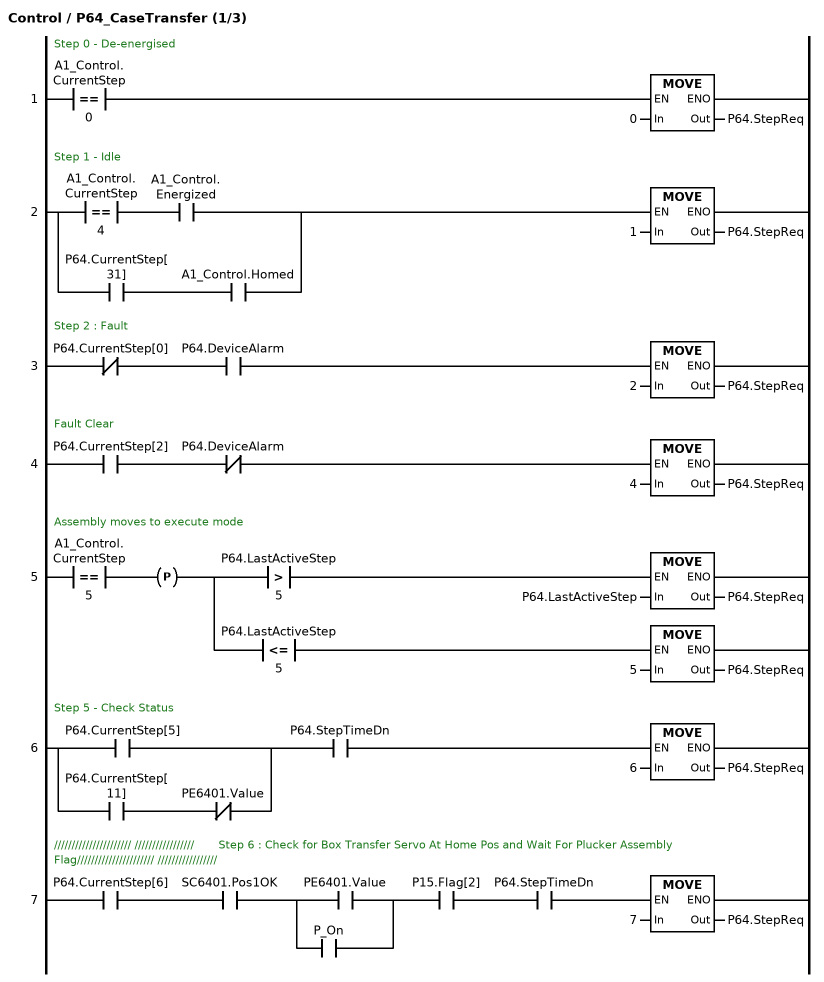
(* [picture p24: Control / P64_CaseTransfer, rungs 1-7] *)
(* Rung 1: Step 0 - De-energised *)
IF A1_Control.CurrentStep = 0 THEN P64.StepReq := 0; END_IF;
(* Rung 2: Step 1 - Idle *)
IF ((A1_Control.CurrentStep = 4) AND A1_Control.Energized) OR (P64.CurrentStep[31] AND A1_Control.Homed) THEN
    P64.StepReq := 1;
END_IF;
(* Rung 3: Step 2 : Fault *)
IF NOT P64.CurrentStep[0] AND P64.DeviceAlarm THEN P64.StepReq := 2; END_IF;
(* Rung 4: Fault Clear *)
IF P64.CurrentStep[2] AND NOT P64.DeviceAlarm THEN P64.StepReq := 4; END_IF;
(* Rung 5: Assembly moves to execute mode *)
_e10(CLK := A1_Control.CurrentStep = 5);
IF _e10.Q AND (P64.LastActiveStep > 5) THEN P64.StepReq := P64.LastActiveStep; END_IF;
IF _e10.Q AND (P64.LastActiveStep <= 5) THEN P64.StepReq := 5; END_IF;
(* Rung 6: Step 5 - Check Status *)
IF (P64.CurrentStep[5] OR (P64.CurrentStep[11] AND NOT PE6401.Value)) AND P64.StepTimeDn THEN
    P64.StepReq := 6;
END_IF;
(* Rung 7: ////////////////////// /////////////////       Step 6 : Check for Box Transfer Servo At Home Pos and Wait For Plucker Assembly Flag////////////////////// ///////////////// *)
IF P64.CurrentStep[6] AND SC6401.Pos1OK AND (PE6401.Value OR P_On) AND P15.Flag[2] AND P64.StepTimeDn THEN
    P64.StepReq := 7;
END_IF;

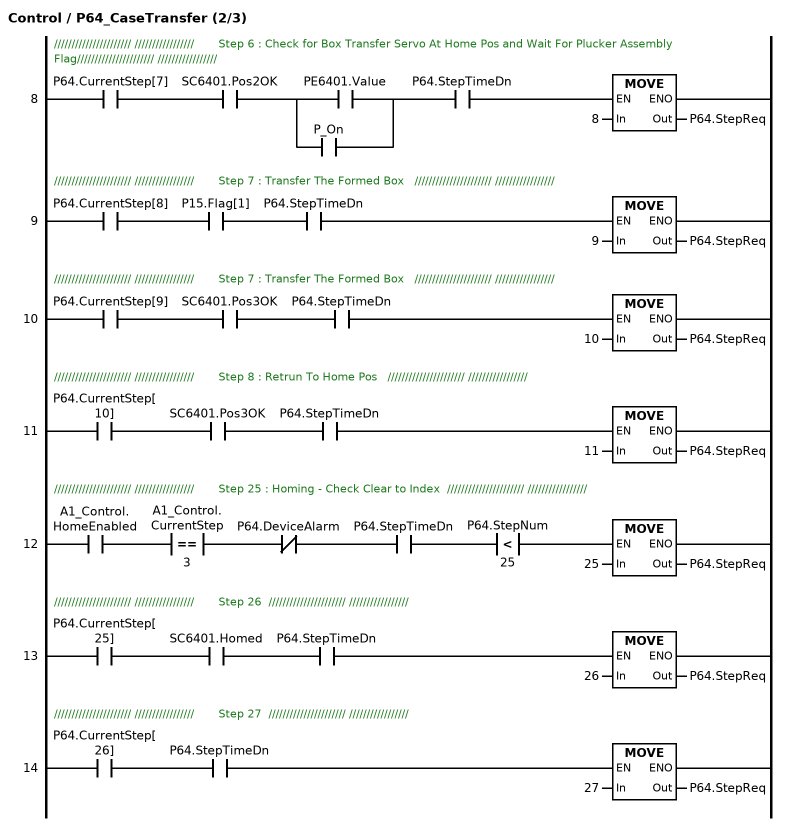
(* Rung 8: ////////////////////// /////////////////       Step 6 : Check for Box Transfer Servo At Home Pos and Wait For Plucker Assembly Flag////////////////////// ///////////////// *)
IF P64.CurrentStep[7] AND SC6401.Pos2OK AND (PE6401.Value OR P_On) AND P64.StepTimeDn THEN
    P64.StepReq := 8;
END_IF;
(* Rung 9: ////////////////////// /////////////////       Step 7 : Transfer The Formed Box   ////////////////////// ///////////////// *)
IF P64.CurrentStep[8] AND P15.Flag[1] AND P64.StepTimeDn THEN P64.StepReq := 9; END_IF;
(* Rung 10: ////////////////////// /////////////////       Step 7 : Transfer The Formed Box   ////////////////////// ///////////////// *)
IF P64.CurrentStep[9] AND SC6401.Pos3OK AND P64.StepTimeDn THEN P64.StepReq := 10; END_IF;
(* Rung 11: ////////////////////// /////////////////       Step 8 : Retrun To Home Pos   ////////////////////// ///////////////// *)
IF P64.CurrentStep[10] AND SC6401.Pos3OK AND P64.StepTimeDn THEN P64.StepReq := 11; END_IF;
(* Rung 12: ////////////////////// /////////////////       Step 25 : Homing - Check Clear to Index  ////////////////////// ///////////////// *)
IF A1_Control.HomeEnabled AND (A1_Control.CurrentStep = 3) AND NOT P64.DeviceAlarm AND P64.StepTimeDn AND (P64.StepNum < 25) THEN
    P64.StepReq := 25;
END_IF;
(* Rung 13: ////////////////////// /////////////////       Step 26  ////////////////////// ///////////////// *)
IF P64.CurrentStep[25] AND SC6401.Homed AND P64.StepTimeDn THEN P64.StepReq := 26; END_IF;
(* Rung 14: ////////////////////// /////////////////       Step 27  ////////////////////// ///////////////// *)
IF P64.CurrentStep[26] AND P64.StepTimeDn THEN P64.StepReq := 27; END_IF;

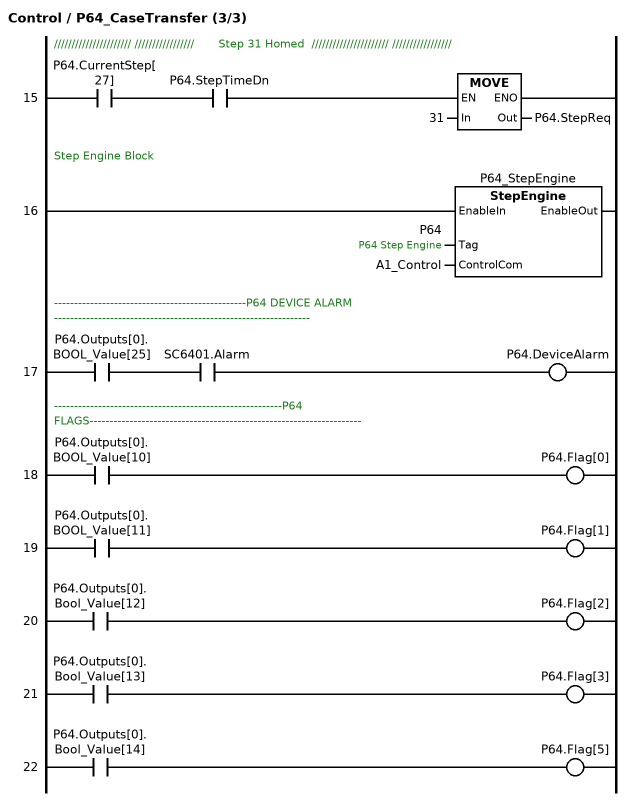
(* Rung 15: ////////////////////// /////////////////       Step 31 Homed  ////////////////////// ///////////////// *)
IF P64.CurrentStep[27] AND P64.StepTimeDn THEN P64.StepReq := 31; END_IF;
(* Rung 16: Step Engine Block *)
P64_StepEngine(EnableIn := TRUE, Tag := P64, ControlCom := A1_Control);
(* Rung 17: ------------------------------------------------P64 DEVICE ALARM ---------------------------------------------------------------- *)
P64.DeviceAlarm := P64.Outputs[0].BOOL_Value[25] AND SC6401.Alarm;
(* Rung 18: ---------------------------------------------------------P64 FLAGS-------------------------------------------------------------------- *)
P64.Flag[0] := P64.Outputs[0].BOOL_Value[10];
(* Rung 19 *)
P64.Flag[1] := P64.Outputs[0].BOOL_Value[11];
(* Rung 20 *)
P64.Flag[2] := P64.Outputs[0].Bool_Value[12];
(* Rung 21 *)
P64.Flag[3] := P64.Outputs[0].Bool_Value[13];
(* Rung 22 *)
P64.Flag[5] := P64.Outputs[0].Bool_Value[14];

(* Section P22_BottomTaping: ladder, written here as Structured Text *)

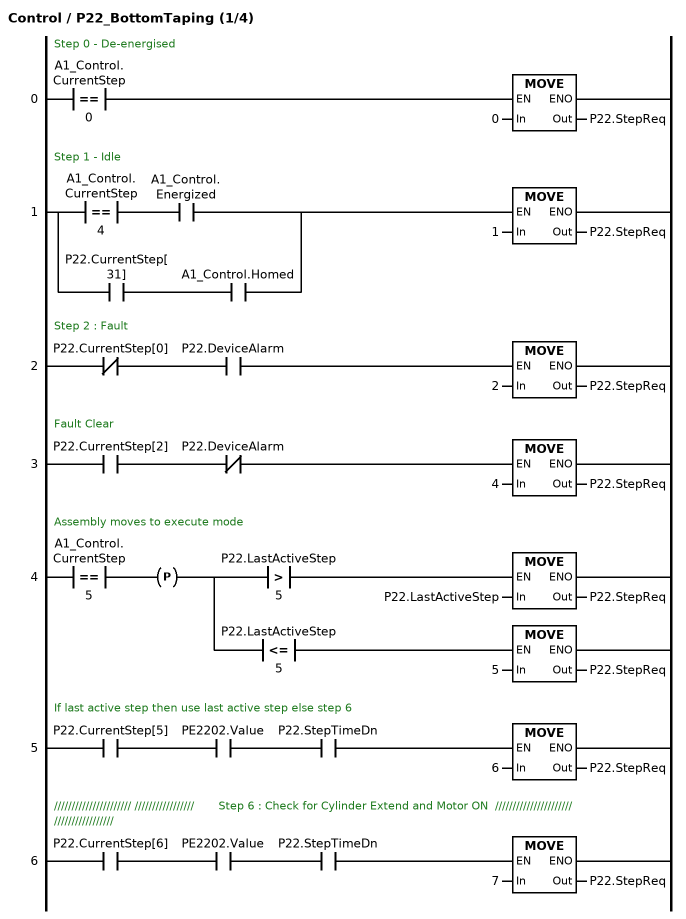
(* Rung 0: Step 0 - De-energised *)
IF A1_Control.CurrentStep = 0 THEN P22.StepReq := 0; END_IF;
(* Rung 1: Step 1 - Idle *)
IF ((A1_Control.CurrentStep = 4) AND A1_Control.Energized) OR (P22.CurrentStep[31] AND A1_Control.Homed) THEN
    P22.StepReq := 1;
END_IF;
(* Rung 2: Step 2 : Fault *)
IF NOT P22.CurrentStep[0] AND P22.DeviceAlarm THEN P22.StepReq := 2; END_IF;
(* Rung 3: Fault Clear *)
IF P22.CurrentStep[2] AND NOT P22.DeviceAlarm THEN P22.StepReq := 4; END_IF;
(* Rung 4: Assembly moves to execute mode *)
_e11(CLK := A1_Control.CurrentStep = 5);
IF _e11.Q AND (P22.LastActiveStep > 5) THEN P22.StepReq := P22.LastActiveStep; END_IF;
IF _e11.Q AND (P22.LastActiveStep <= 5) THEN P22.StepReq := 5; END_IF;
(* Rung 5: If last active step then use last active step else step 6 *)
IF P22.CurrentStep[5] AND PE2202.Value AND P22.StepTimeDn THEN P22.StepReq := 6; END_IF;
(* Rung 6: ////////////////////// /////////////////       Step 6 : Check for Cylinder Extend and Motor ON  ////////////////////// ///////////////// *)
IF P22.CurrentStep[6] AND PE2202.Value AND P22.StepTimeDn THEN P22.StepReq := 7; END_IF;

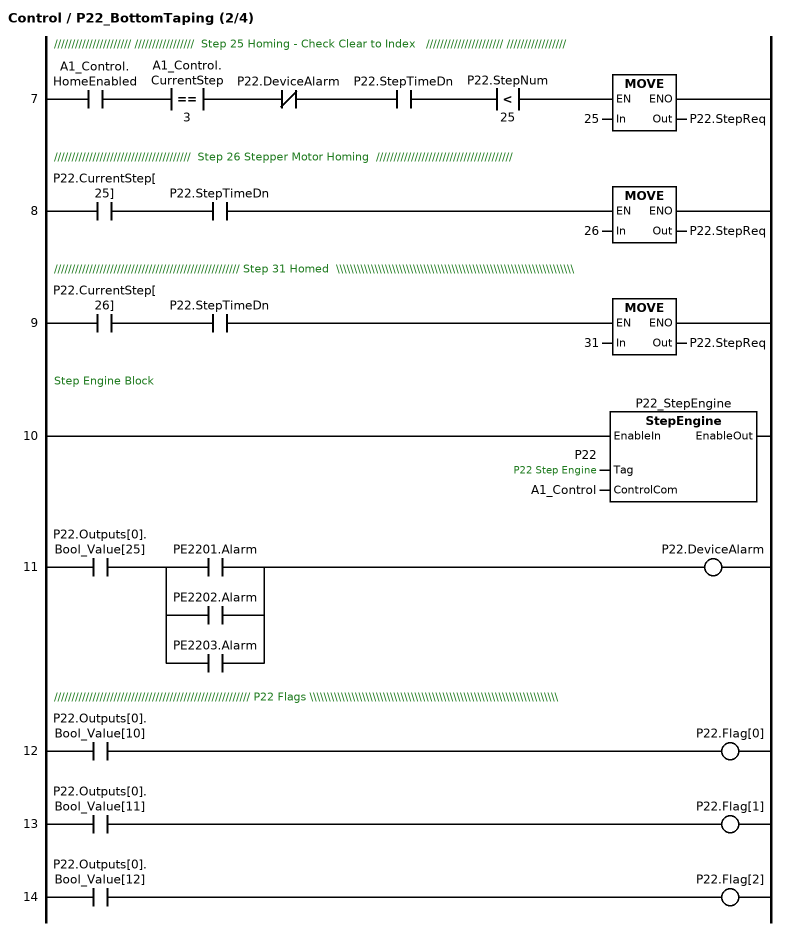
(* Rung 7: ////////////////////// /////////////////  Step 25 Homing - Check Clear to Index   ////////////////////// ///////////////// *)
IF A1_Control.HomeEnabled AND (A1_Control.CurrentStep = 3) AND NOT P22.DeviceAlarm AND P22.StepTimeDn AND (P22.StepNum < 25) THEN
    P22.StepReq := 25;
END_IF;
(* Rung 8: ///////////////////////////////////////  Step 26 Stepper Motor Homing  /////////////////////////////////////// *)
IF P22.CurrentStep[25] AND P22.StepTimeDn THEN P22.StepReq := 26; END_IF;
(* Rung 9: ///////////////////////////////////////////////////// Step 31 Homed  \\\\\\\\\\\\\\\\\\\\\\\\\\\\\\\\\\\\\\\\\\\\\\\\\\\\\\\\\\\\\\\\\\\\ *)
IF P22.CurrentStep[26] AND P22.StepTimeDn THEN P22.StepReq := 31; END_IF;
(* Rung 10: Step Engine Block *)
P22_StepEngine(EnableIn := TRUE, Tag := P22, ControlCom := A1_Control);
(* Rung 11 *)
P22.DeviceAlarm := P22.Outputs[0].Bool_Value[25] AND (PE2201.Alarm OR PE2202.Alarm OR PE2203.Alarm);
(* Rung 12: //////////////////////////////////////////////////////// P22 Flags \\\\\\\\\\\\\\\\\\\\\\\\\\\\\\\\\\\\\\\\\\\\\\\\\\\\\\\\\\\\\\\\\\\\\\\ *)
P22.Flag[0] := P22.Outputs[0].Bool_Value[10];
(* Rung 13 *)
P22.Flag[1] := P22.Outputs[0].Bool_Value[11];
(* Rung 14 *)
P22.Flag[2] := P22.Outputs[0].Bool_Value[12];

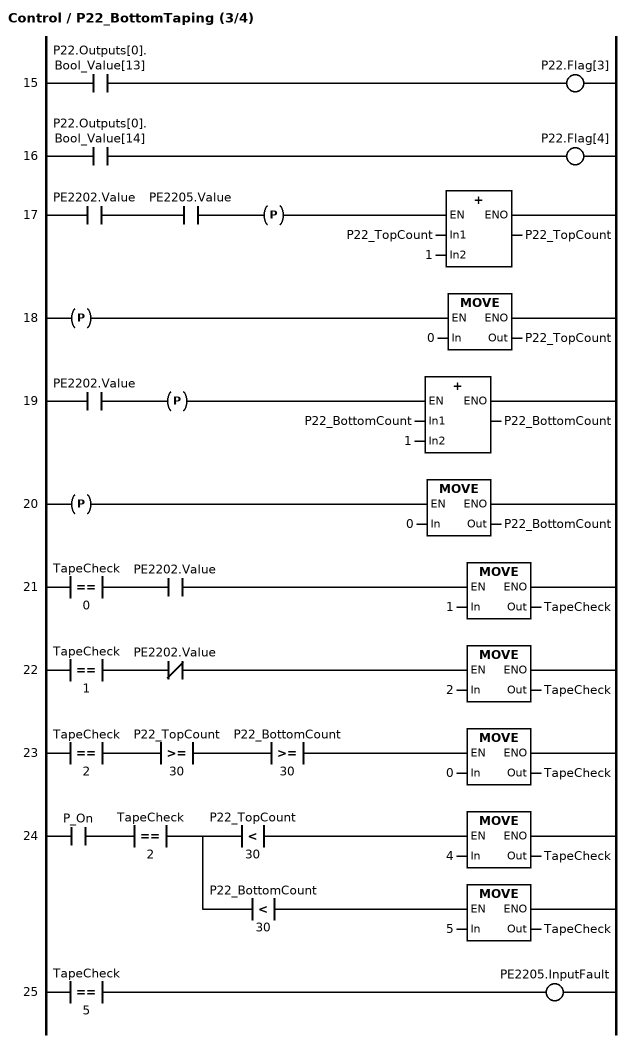
(* Rung 15 *)
P22.Flag[3] := P22.Outputs[0].Bool_Value[13];
(* Rung 16 *)
P22.Flag[4] := P22.Outputs[0].Bool_Value[14];
(* Rung 17 *)
_e12(CLK := PE2202.Value AND PE2205.Value);
IF _e12.Q THEN P22_TopCount := P22_TopCount + 1; END_IF;
(* Rung 18 *)
_e13(CLK := TRUE);
IF _e13.Q THEN P22_TopCount := 0; END_IF;
(* Rung 19 *)
_e14(CLK := PE2202.Value);
IF _e14.Q THEN P22_BottomCount := P22_BottomCount + 1; END_IF;
(* Rung 20 *)
_e15(CLK := TRUE);
IF _e15.Q THEN P22_BottomCount := 0; END_IF;
(* Rung 21 *)
IF (TapeCheck = 0) AND PE2202.Value THEN TapeCheck := 1; END_IF;
(* Rung 22 *)
IF (TapeCheck = 1) AND NOT PE2202.Value THEN TapeCheck := 2; END_IF;
(* Rung 23 *)
IF (TapeCheck = 2) AND (P22_TopCount >= 30) AND (P22_BottomCount >= 30) THEN TapeCheck := 0; END_IF;
(* Rung 24 *)
_p16 := P_On AND (TapeCheck = 2);
IF P_On AND (TapeCheck = 2) AND (P22_TopCount < 30) THEN TapeCheck := 4; END_IF;
IF _p16 AND (P22_BottomCount < 30) THEN TapeCheck := 5; END_IF;
(* Rung 25 *)
PE2205.InputFault := TapeCheck = 5;

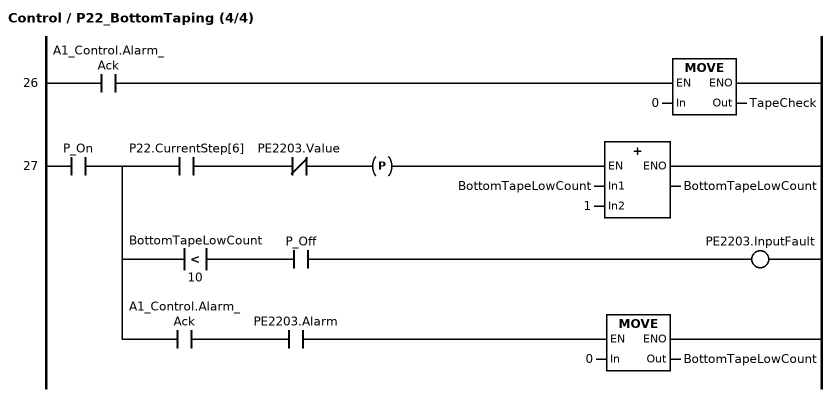
(* Rung 26 *)
IF A1_Control.Alarm_Ack THEN TapeCheck := 0; END_IF;
(* Rung 27 *)
_e17(CLK := P_On AND P22.CurrentStep[6] AND NOT PE2203.Value);
IF _e17.Q THEN BottomTapeLowCount := BottomTapeLowCount + 1; END_IF;
PE2203.InputFault := P_On AND (BottomTapeLowCount < 10) AND P_Off;
IF P_On AND A1_Control.Alarm_Ack AND PE2203.Alarm THEN BottomTapeLowCount := 0; END_IF;

(* Section P18_InfeedConveyor_1: ladder, written here as Structured Text *)

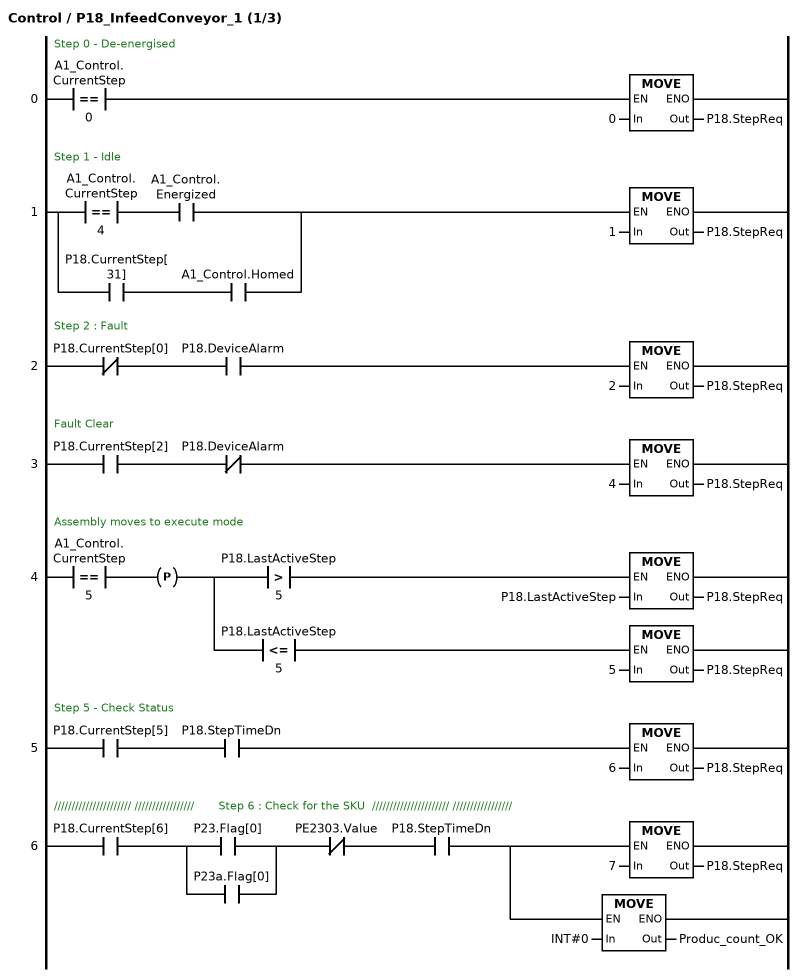
(* Rung 0: Step 0 - De-energised *)
IF A1_Control.CurrentStep = 0 THEN P18.StepReq := 0; END_IF;
(* Rung 1: Step 1 - Idle *)
IF ((A1_Control.CurrentStep = 4) AND A1_Control.Energized) OR (P18.CurrentStep[31] AND A1_Control.Homed) THEN
    P18.StepReq := 1;
END_IF;
(* Rung 2: Step 2 : Fault *)
IF NOT P18.CurrentStep[0] AND P18.DeviceAlarm THEN P18.StepReq := 2; END_IF;
(* Rung 3: Fault Clear *)
IF P18.CurrentStep[2] AND NOT P18.DeviceAlarm THEN P18.StepReq := 4; END_IF;
(* Rung 4: Assembly moves to execute mode *)
_e18(CLK := A1_Control.CurrentStep = 5);
IF _e18.Q AND (P18.LastActiveStep > 5) THEN P18.StepReq := P18.LastActiveStep; END_IF;
IF _e18.Q AND (P18.LastActiveStep <= 5) THEN P18.StepReq := 5; END_IF;
(* Rung 5: Step 5 - Check Status *)
IF P18.CurrentStep[5] AND P18.StepTimeDn THEN P18.StepReq := 6; END_IF;
(* Rung 6: ////////////////////// /////////////////       Step 6 : Check for the SKU  ////////////////////// ///////////////// *)
_p19 := P18.CurrentStep[6] AND (P23.Flag[0] OR P23a.Flag[0]) AND NOT PE2303.Value AND P18.StepTimeDn;
IF _p19 THEN
    P18.StepReq := 7;
    Produc_count_OK := INT#0;
END_IF;

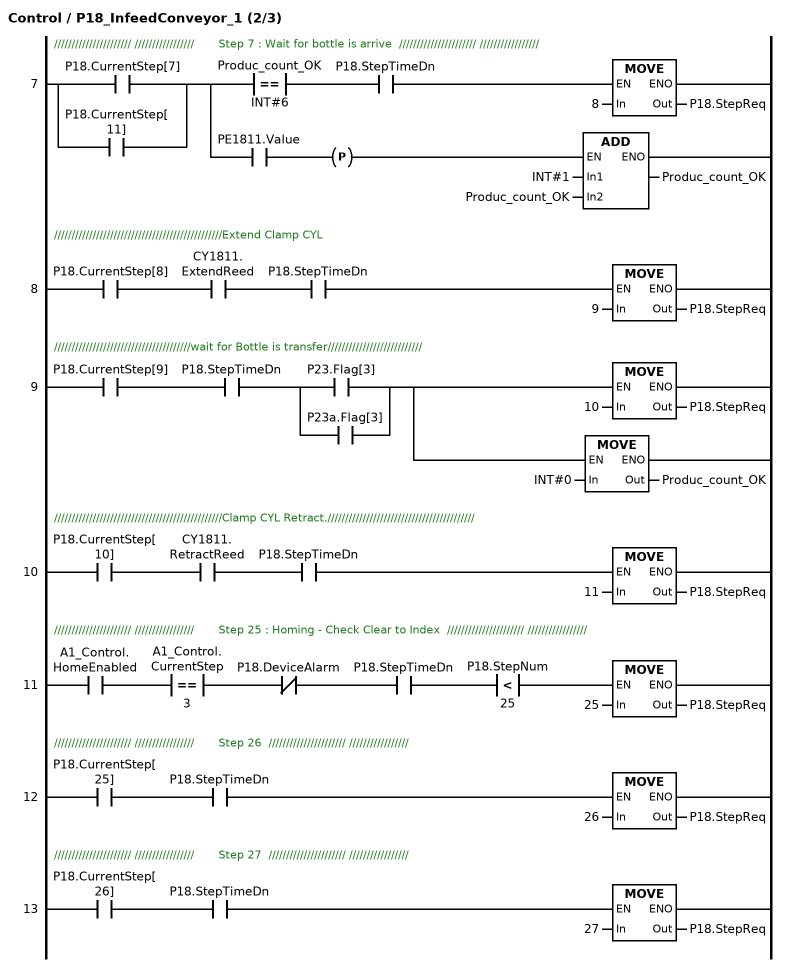
(* Rung 7: ////////////////////// /////////////////       Step 7 : Wait for bottle is arrive  ////////////////////// ///////////////// *)
_p20 := P18.CurrentStep[7] OR P18.CurrentStep[11];
IF (P18.CurrentStep[7] OR P18.CurrentStep[11]) AND (Produc_count_OK = INT#6) AND P18.StepTimeDn THEN
    P18.StepReq := 8;
END_IF;
_e21(CLK := _p20 AND PE1811.Value);
IF _e21.Q THEN Produc_count_OK := INT#1 + Produc_count_OK; END_IF;
(* Rung 8: ////////////////////////////////////////////////Extend Clamp CYL *)
IF P18.CurrentStep[8] AND CY1811.ExtendReed AND P18.StepTimeDn THEN P18.StepReq := 9; END_IF;
(* Rung 9: ///////////////////////////////////////wait for Bottle is transfer/////////////////////////// *)
_p22 := P18.CurrentStep[9] AND P18.StepTimeDn AND (P23.Flag[3] OR P23a.Flag[3]);
IF _p22 THEN
    P18.StepReq := 10;
    Produc_count_OK := INT#0;
END_IF;
(* Rung 10: ////////////////////////////////////////////////Clamp CYL Retract.////////////////////////////////////////// *)
IF P18.CurrentStep[10] AND CY1811.RetractReed AND P18.StepTimeDn THEN P18.StepReq := 11; END_IF;
(* Rung 11: ////////////////////// /////////////////       Step 25 : Homing - Check Clear to Index  ////////////////////// ///////////////// *)
IF A1_Control.HomeEnabled AND (A1_Control.CurrentStep = 3) AND NOT P18.DeviceAlarm AND P18.StepTimeDn AND (P18.StepNum < 25) THEN
    P18.StepReq := 25;
END_IF;
(* Rung 12: ////////////////////// /////////////////       Step 26  ////////////////////// ///////////////// *)
IF P18.CurrentStep[25] AND P18.StepTimeDn THEN P18.StepReq := 26; END_IF;
(* Rung 13: ////////////////////// /////////////////       Step 27  ////////////////////// ///////////////// *)
IF P18.CurrentStep[26] AND P18.StepTimeDn THEN P18.StepReq := 27; END_IF;

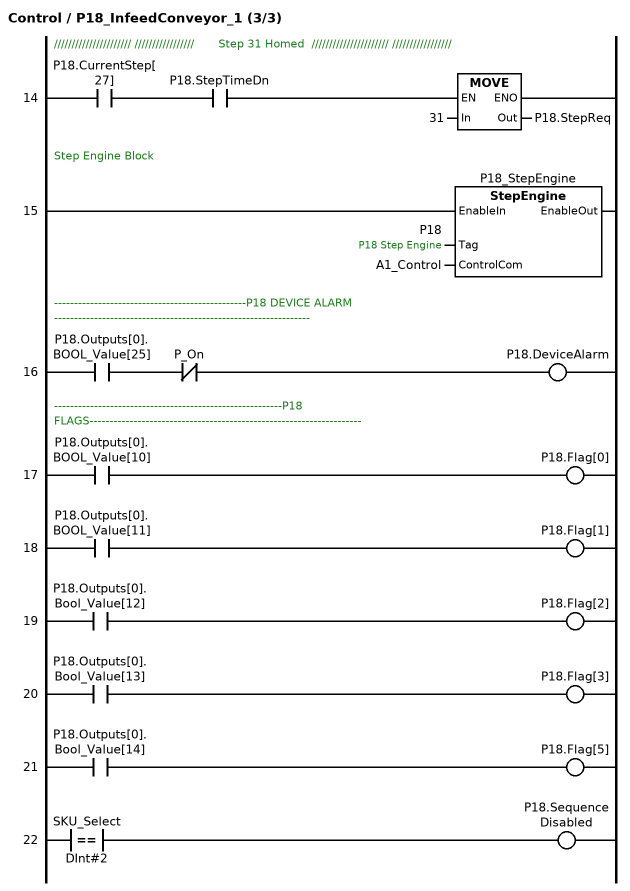
(* Rung 14: ////////////////////// /////////////////       Step 31 Homed  ////////////////////// ///////////////// *)
IF P18.CurrentStep[27] AND P18.StepTimeDn THEN P18.StepReq := 31; END_IF;
(* Rung 15: Step Engine Block *)
P18_StepEngine(EnableIn := TRUE, Tag := P18, ControlCom := A1_Control);
(* Rung 16: ------------------------------------------------P18 DEVICE ALARM ---------------------------------------------------------------- *)
P18.DeviceAlarm := P18.Outputs[0].BOOL_Value[25] AND NOT P_On;
(* Rung 17: ---------------------------------------------------------P18 FLAGS-------------------------------------------------------------------- *)
P18.Flag[0] := P18.Outputs[0].BOOL_Value[10];
(* Rung 18 *)
P18.Flag[1] := P18.Outputs[0].BOOL_Value[11];
(* Rung 19 *)
P18.Flag[2] := P18.Outputs[0].Bool_Value[12];
(* Rung 20 *)
P18.Flag[3] := P18.Outputs[0].Bool_Value[13];
(* Rung 21 *)
P18.Flag[5] := P18.Outputs[0].Bool_Value[14];
(* Rung 22 *)
P18.SequenceDisabled := SKU_Select = DInt#2;

(* Section P28_layerBoard: ladder, written here as Structured Text *)

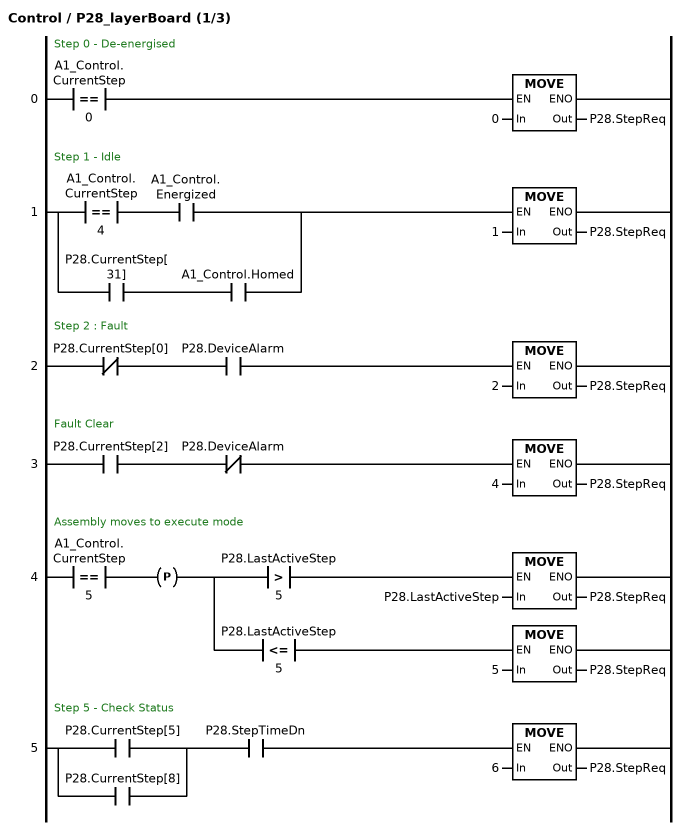
(* Rung 0: Step 0 - De-energised *)
IF A1_Control.CurrentStep = 0 THEN P28.StepReq := 0; END_IF;
(* Rung 1: Step 1 - Idle *)
IF ((A1_Control.CurrentStep = 4) AND A1_Control.Energized) OR (P28.CurrentStep[31] AND A1_Control.Homed) THEN
    P28.StepReq := 1;
END_IF;
(* Rung 2: Step 2 : Fault *)
IF NOT P28.CurrentStep[0] AND P28.DeviceAlarm THEN P28.StepReq := 2; END_IF;
(* Rung 3: Fault Clear *)
IF P28.CurrentStep[2] AND NOT P28.DeviceAlarm THEN P28.StepReq := 4; END_IF;
(* Rung 4: Assembly moves to execute mode *)
_e23(CLK := A1_Control.CurrentStep = 5);
IF _e23.Q AND (P28.LastActiveStep > 5) THEN P28.StepReq := P28.LastActiveStep; END_IF;
IF _e23.Q AND (P28.LastActiveStep <= 5) THEN P28.StepReq := 5; END_IF;
(* Rung 5: Step 5 - Check Status *)
IF (P28.CurrentStep[5] OR P28.CurrentStep[8]) AND P28.StepTimeDn THEN P28.StepReq := 6; END_IF;

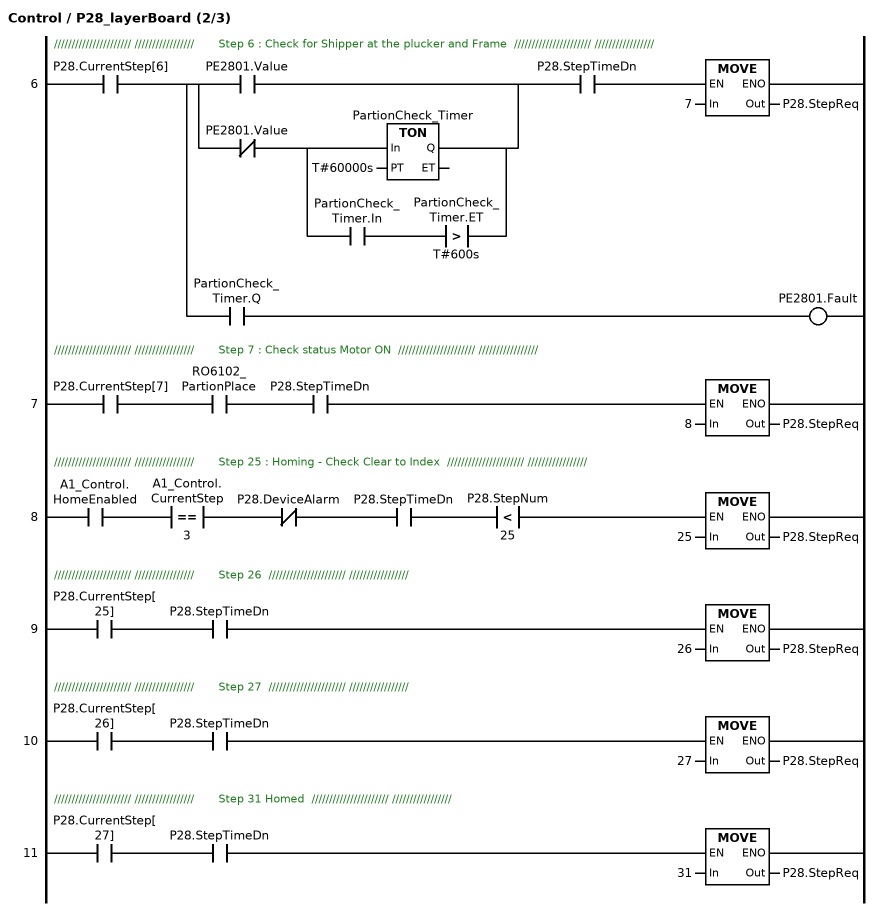
(* Rung 6: ////////////////////// /////////////////       Step 6 : Check for Shipper at the plucker and Frame  ////////////////////// ///////////////// *)
PartionCheck_Timer(In := P28.CurrentStep[6] AND NOT PE2801.Value, PT := T#60000s);
_p24 := P28.CurrentStep[6];
IF ((P28.CurrentStep[6] AND PE2801.Value) OR PartionCheck_Timer.Q OR (P28.CurrentStep[6] AND NOT PE2801.Value AND PartionCheck_Timer.In AND (PartionCheck_Timer.ET > T#600s))) AND P28.StepTimeDn THEN
    P28.StepReq := 7;
END_IF;
PE2801.Fault := _p24 AND PartionCheck_Timer.Q;
(* Rung 7: ////////////////////// /////////////////       Step 7 : Check status Motor ON  ////////////////////// ///////////////// *)
IF P28.CurrentStep[7] AND RO6102_PartionPlace AND P28.StepTimeDn THEN P28.StepReq := 8; END_IF;
(* Rung 8: ////////////////////// /////////////////       Step 25 : Homing - Check Clear to Index  ////////////////////// ///////////////// *)
IF A1_Control.HomeEnabled AND (A1_Control.CurrentStep = 3) AND NOT P28.DeviceAlarm AND P28.StepTimeDn AND (P28.StepNum < 25) THEN
    P28.StepReq := 25;
END_IF;
(* Rung 9: ////////////////////// /////////////////       Step 26  ////////////////////// ///////////////// *)
IF P28.CurrentStep[25] AND P28.StepTimeDn THEN P28.StepReq := 26; END_IF;
(* Rung 10: ////////////////////// /////////////////       Step 27  ////////////////////// ///////////////// *)
IF P28.CurrentStep[26] AND P28.StepTimeDn THEN P28.StepReq := 27; END_IF;
(* Rung 11: ////////////////////// /////////////////       Step 31 Homed  ////////////////////// ///////////////// *)
IF P28.CurrentStep[27] AND P28.StepTimeDn THEN P28.StepReq := 31; END_IF;

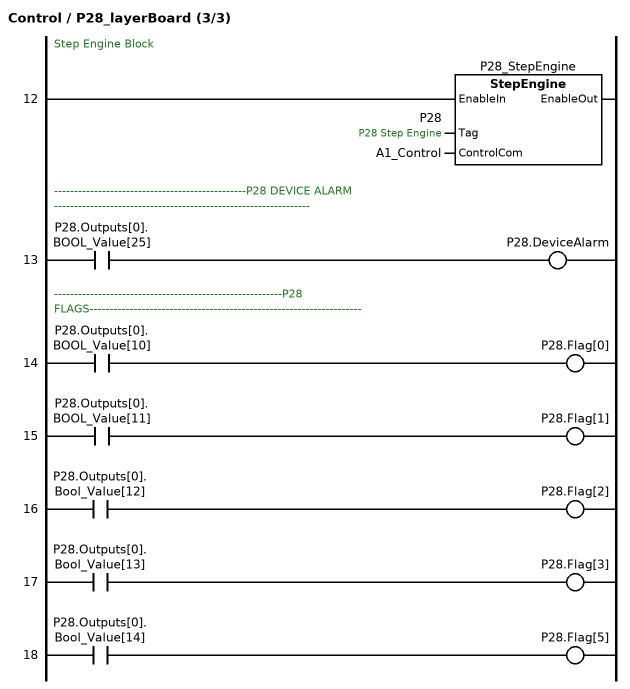
(* Rung 12: Step Engine Block *)
P28_StepEngine(EnableIn := TRUE, Tag := P28, ControlCom := A1_Control);
(* Rung 13: ------------------------------------------------P28 DEVICE ALARM ---------------------------------------------------------------- *)
P28.DeviceAlarm := P28.Outputs[0].BOOL_Value[25];
(* Rung 14: ---------------------------------------------------------P28 FLAGS-------------------------------------------------------------------- *)
P28.Flag[0] := P28.Outputs[0].BOOL_Value[10];
(* Rung 15 *)
P28.Flag[1] := P28.Outputs[0].BOOL_Value[11];
(* Rung 16 *)
P28.Flag[2] := P28.Outputs[0].Bool_Value[12];
(* Rung 17 *)
P28.Flag[3] := P28.Outputs[0].Bool_Value[13];
(* Rung 18 *)
P28.Flag[5] := P28.Outputs[0].Bool_Value[14];

(* Section P18a_InfeedConveyor_2: ladder, written here as Structured Text *)

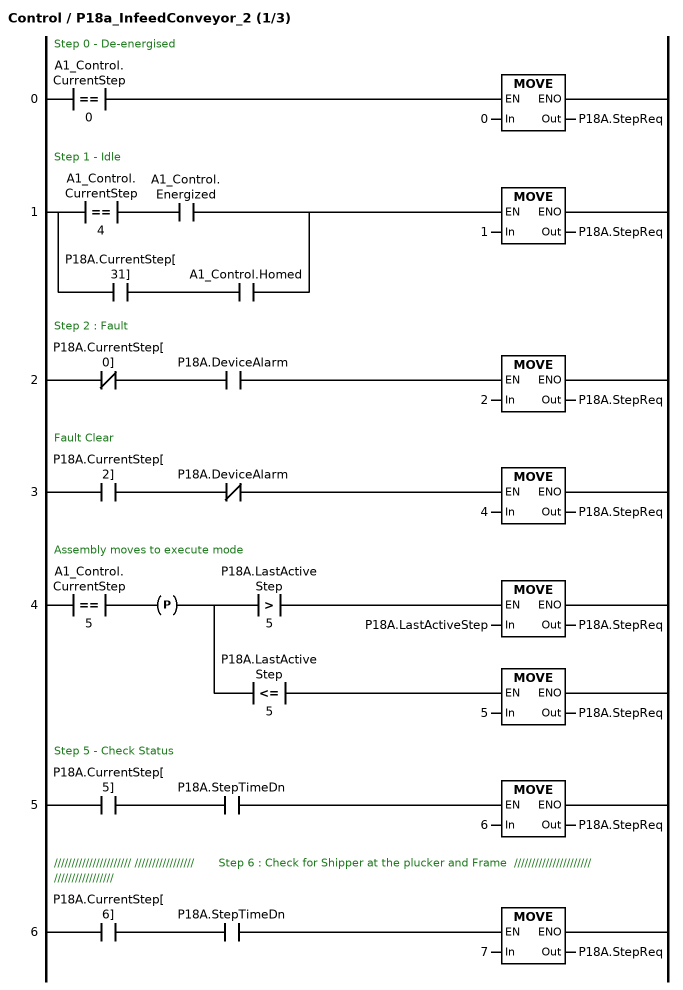
(* Rung 0: Step 0 - De-energised *)
IF A1_Control.CurrentStep = 0 THEN P18A.StepReq := 0; END_IF;
(* Rung 1: Step 1 - Idle *)
IF ((A1_Control.CurrentStep = 4) AND A1_Control.Energized) OR (P18A.CurrentStep[31] AND A1_Control.Homed) THEN
    P18A.StepReq := 1;
END_IF;
(* Rung 2: Step 2 : Fault *)
IF NOT P18A.CurrentStep[0] AND P18A.DeviceAlarm THEN P18A.StepReq := 2; END_IF;
(* Rung 3: Fault Clear *)
IF P18A.CurrentStep[2] AND NOT P18A.DeviceAlarm THEN P18A.StepReq := 4; END_IF;
(* Rung 4: Assembly moves to execute mode *)
_e25(CLK := A1_Control.CurrentStep = 5);
IF _e25.Q AND (P18A.LastActiveStep > 5) THEN P18A.StepReq := P18A.LastActiveStep; END_IF;
IF _e25.Q AND (P18A.LastActiveStep <= 5) THEN P18A.StepReq := 5; END_IF;
(* Rung 5: Step 5 - Check Status *)
IF P18A.CurrentStep[5] AND P18A.StepTimeDn THEN P18A.StepReq := 6; END_IF;
(* Rung 6: ////////////////////// /////////////////       Step 6 : Check for Shipper at the plucker and Frame  ////////////////////// ///////////////// *)
IF P18A.CurrentStep[6] AND P18A.StepTimeDn THEN P18A.StepReq := 7; END_IF;

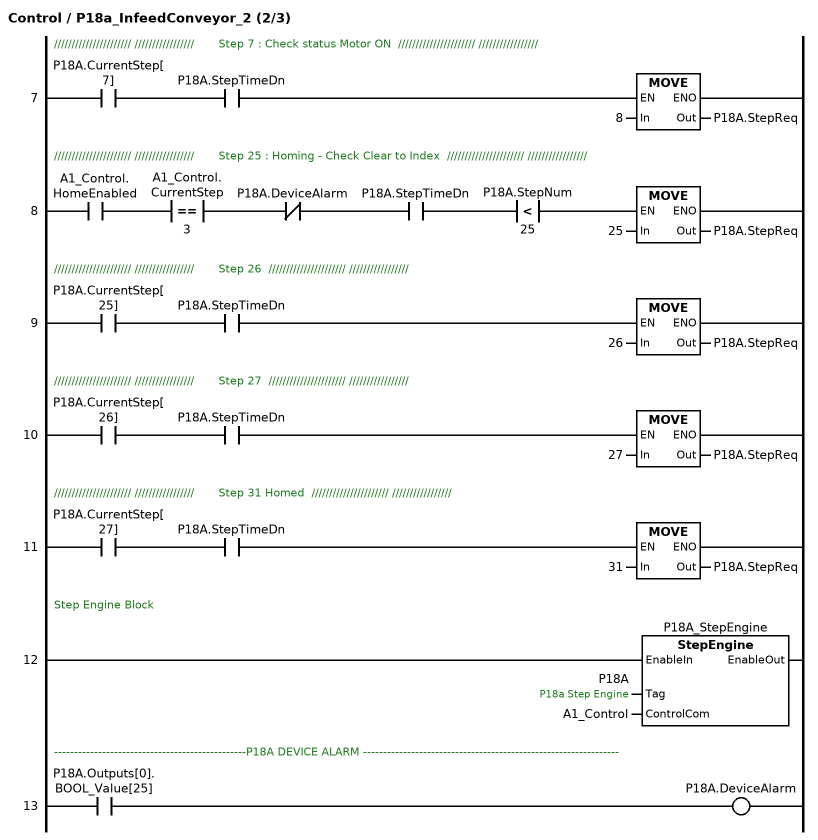
(* Rung 7: ////////////////////// /////////////////       Step 7 : Check status Motor ON  ////////////////////// ///////////////// *)
IF P18A.CurrentStep[7] AND P18A.StepTimeDn THEN P18A.StepReq := 8; END_IF;
(* Rung 8: ////////////////////// /////////////////       Step 25 : Homing - Check Clear to Index  ////////////////////// ///////////////// *)
IF A1_Control.HomeEnabled AND (A1_Control.CurrentStep = 3) AND NOT P18A.DeviceAlarm AND P18A.StepTimeDn AND (P18A.StepNum < 25) THEN
    P18A.StepReq := 25;
END_IF;
(* Rung 9: ////////////////////// /////////////////       Step 26  ////////////////////// ///////////////// *)
IF P18A.CurrentStep[25] AND P18A.StepTimeDn THEN P18A.StepReq := 26; END_IF;
(* Rung 10: ////////////////////// /////////////////       Step 27  ////////////////////// ///////////////// *)
IF P18A.CurrentStep[26] AND P18A.StepTimeDn THEN P18A.StepReq := 27; END_IF;
(* Rung 11: ////////////////////// /////////////////       Step 31 Homed  ////////////////////// ///////////////// *)
IF P18A.CurrentStep[27] AND P18A.StepTimeDn THEN P18A.StepReq := 31; END_IF;
(* Rung 12: Step Engine Block *)
P18A_StepEngine(EnableIn := TRUE, Tag := P18A, ControlCom := A1_Control);
(* Rung 13: ------------------------------------------------P18A DEVICE ALARM ---------------------------------------------------------------- *)
P18A.DeviceAlarm := P18A.Outputs[0].BOOL_Value[25];

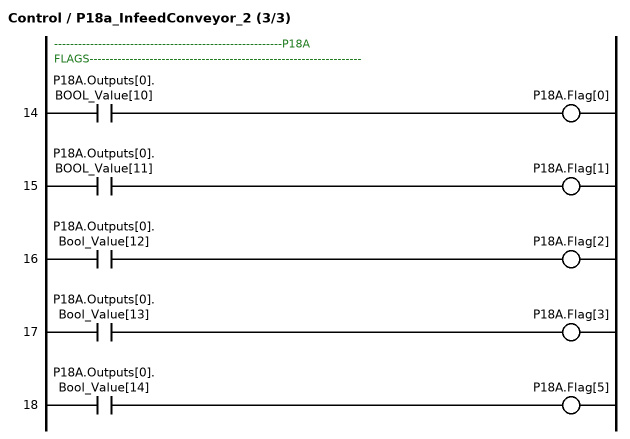
(* Rung 14: ---------------------------------------------------------P18A FLAGS-------------------------------------------------------------------- *)
P18A.Flag[0] := P18A.Outputs[0].BOOL_Value[10];
(* Rung 15 *)
P18A.Flag[1] := P18A.Outputs[0].BOOL_Value[11];
(* Rung 16 *)
P18A.Flag[2] := P18A.Outputs[0].Bool_Value[12];
(* Rung 17 *)
P18A.Flag[3] := P18A.Outputs[0].Bool_Value[13];
(* Rung 18 *)
P18A.Flag[5] := P18A.Outputs[0].Bool_Value[14];

(* Section P23_Collation_Unit_1: ladder, written here as Structured Text *)

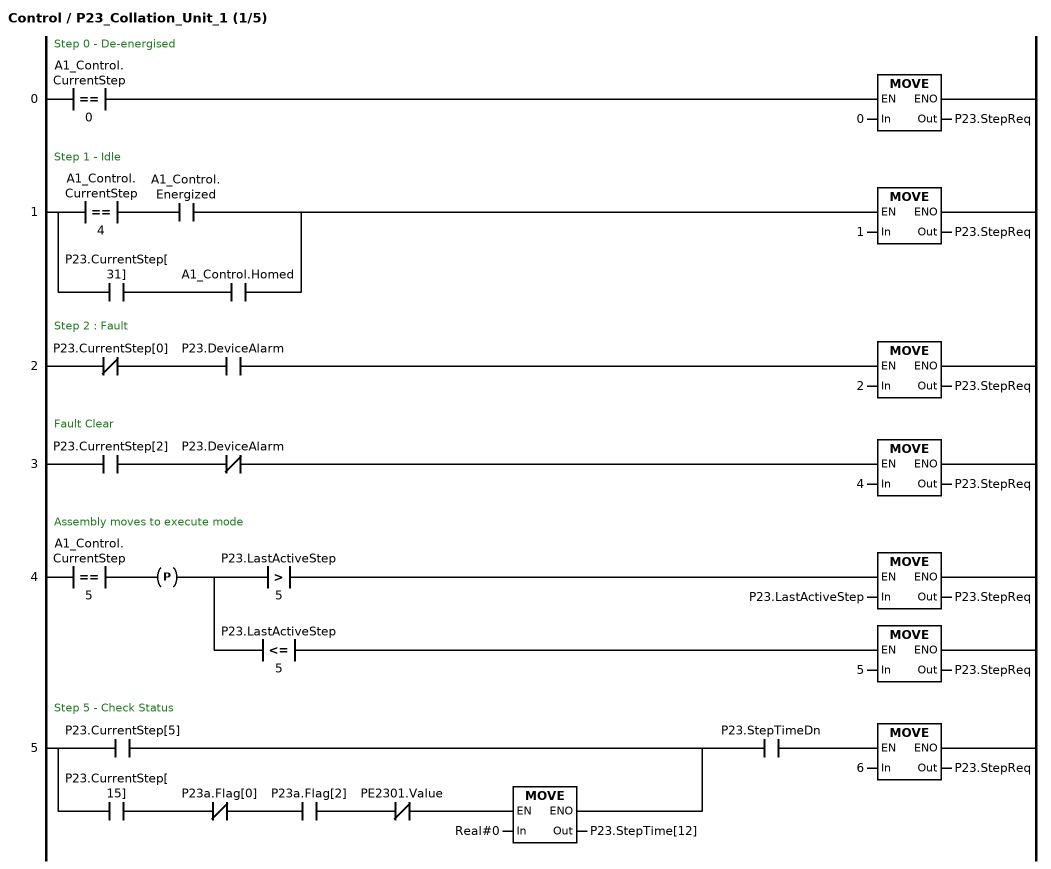
(* Rung 0: Step 0 - De-energised *)
IF A1_Control.CurrentStep = 0 THEN P23.StepReq := 0; END_IF;
(* Rung 1: Step 1 - Idle *)
IF ((A1_Control.CurrentStep = 4) AND A1_Control.Energized) OR (P23.CurrentStep[31] AND A1_Control.Homed) THEN
    P23.StepReq := 1;
END_IF;
(* Rung 2: Step 2 : Fault *)
IF NOT P23.CurrentStep[0] AND P23.DeviceAlarm THEN P23.StepReq := 2; END_IF;
(* Rung 3: Fault Clear *)
IF P23.CurrentStep[2] AND NOT P23.DeviceAlarm THEN P23.StepReq := 4; END_IF;
(* Rung 4: Assembly moves to execute mode *)
_e26(CLK := A1_Control.CurrentStep = 5);
IF _e26.Q AND (P23.LastActiveStep > 5) THEN P23.StepReq := P23.LastActiveStep; END_IF;
IF _e26.Q AND (P23.LastActiveStep <= 5) THEN P23.StepReq := 5; END_IF;
(* Rung 5: Step 5 - Check Status *)
_p27 := P23.CurrentStep[5];
_p28 := P23.CurrentStep[15] AND NOT P23a.Flag[0] AND P23a.Flag[2] AND NOT PE2301.Value;
IF _p28 THEN P23.StepTime[12] := Real#0; END_IF;
IF (_p27 OR _p28) AND P23.StepTimeDn THEN P23.StepReq := 6; END_IF;

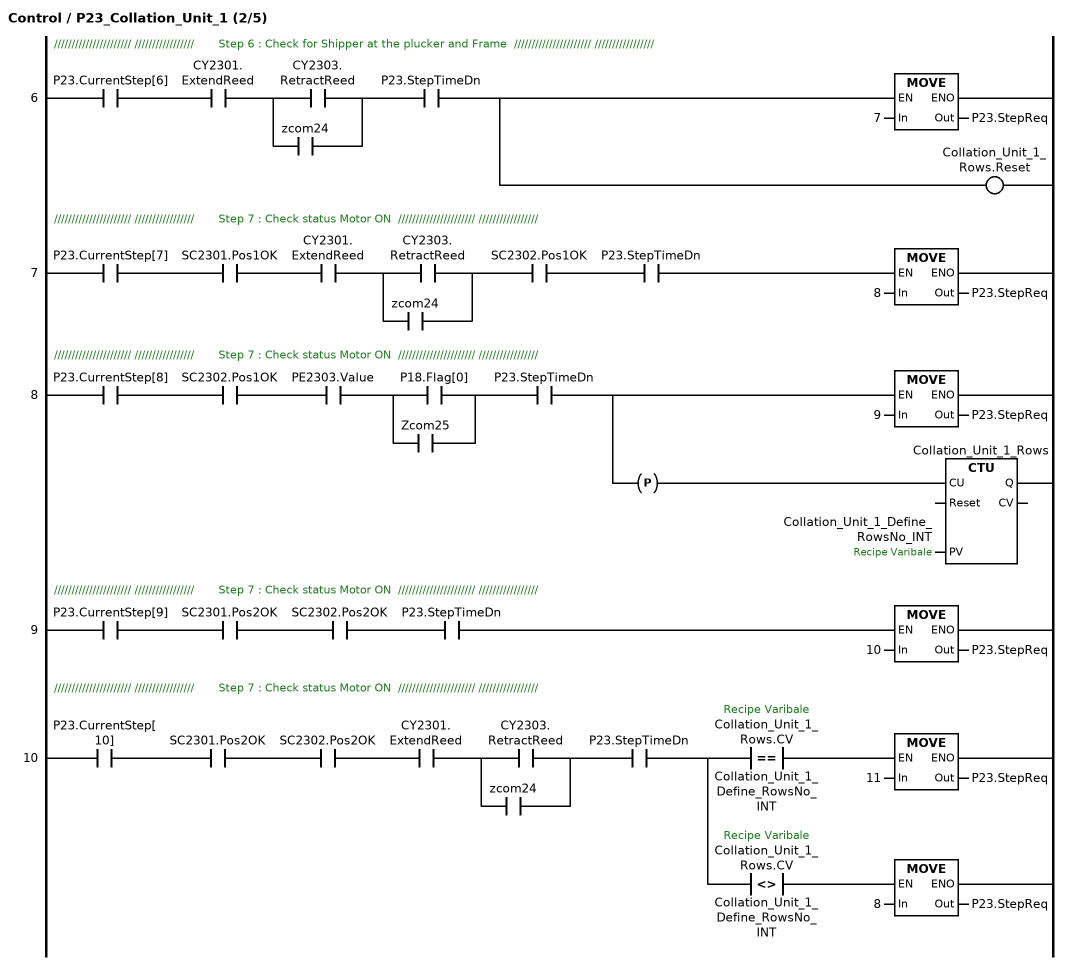
(* Rung 6: ////////////////////// /////////////////       Step 6 : Check for Shipper at the plucker and Frame  ////////////////////// ///////////////// *)
_p29 := P23.CurrentStep[6] AND CY2301.ExtendReed AND (CY2303.RetractReed OR zcom24) AND P23.StepTimeDn;
IF _p29 THEN P23.StepReq := 7; END_IF;
Collation_Unit_1_Rows.Reset := _p29;
(* Rung 7: ////////////////////// /////////////////       Step 7 : Check status Motor ON  ////////////////////// ///////////////// *)
IF P23.CurrentStep[7] AND SC2301.Pos1OK AND CY2301.ExtendReed AND (CY2303.RetractReed OR zcom24) AND SC2302.Pos1OK AND P23.StepTimeDn THEN
    P23.StepReq := 8;
END_IF;
(* Rung 8: ////////////////////// /////////////////       Step 7 : Check status Motor ON  ////////////////////// ///////////////// *)
_p30 := P23.CurrentStep[8] AND SC2302.Pos1OK AND PE2303.Value AND (P18.Flag[0] OR Zcom25) AND P23.StepTimeDn;
IF _p30 THEN P23.StepReq := 9; END_IF;
_e31(CLK := _p30);
_e32(CLK := _e31.Q);
Collation_Unit_1_Rows(CU := _e32.Q, PV := Collation_Unit_1_Define_RowsNo_INT);
(* Rung 9: ////////////////////// /////////////////       Step 7 : Check status Motor ON  ////////////////////// ///////////////// *)
IF P23.CurrentStep[9] AND SC2301.Pos2OK AND SC2302.Pos2OK AND P23.StepTimeDn THEN
    P23.StepReq := 10;
END_IF;
(* Rung 10: ////////////////////// /////////////////       Step 7 : Check status Motor ON  ////////////////////// ///////////////// *)
_p33 := P23.CurrentStep[10] AND SC2301.Pos2OK AND SC2302.Pos2OK AND CY2301.ExtendReed AND (CY2303.RetractReed OR zcom24) AND P23.StepTimeDn;
IF _p33 AND (Collation_Unit_1_Rows.CV = Collation_Unit_1_Define_RowsNo_INT) THEN
    P23.StepReq := 11;
END_IF;
IF _p33 AND (Collation_Unit_1_Rows.CV <> Collation_Unit_1_Define_RowsNo_INT) THEN
    P23.StepReq := 8;
END_IF;

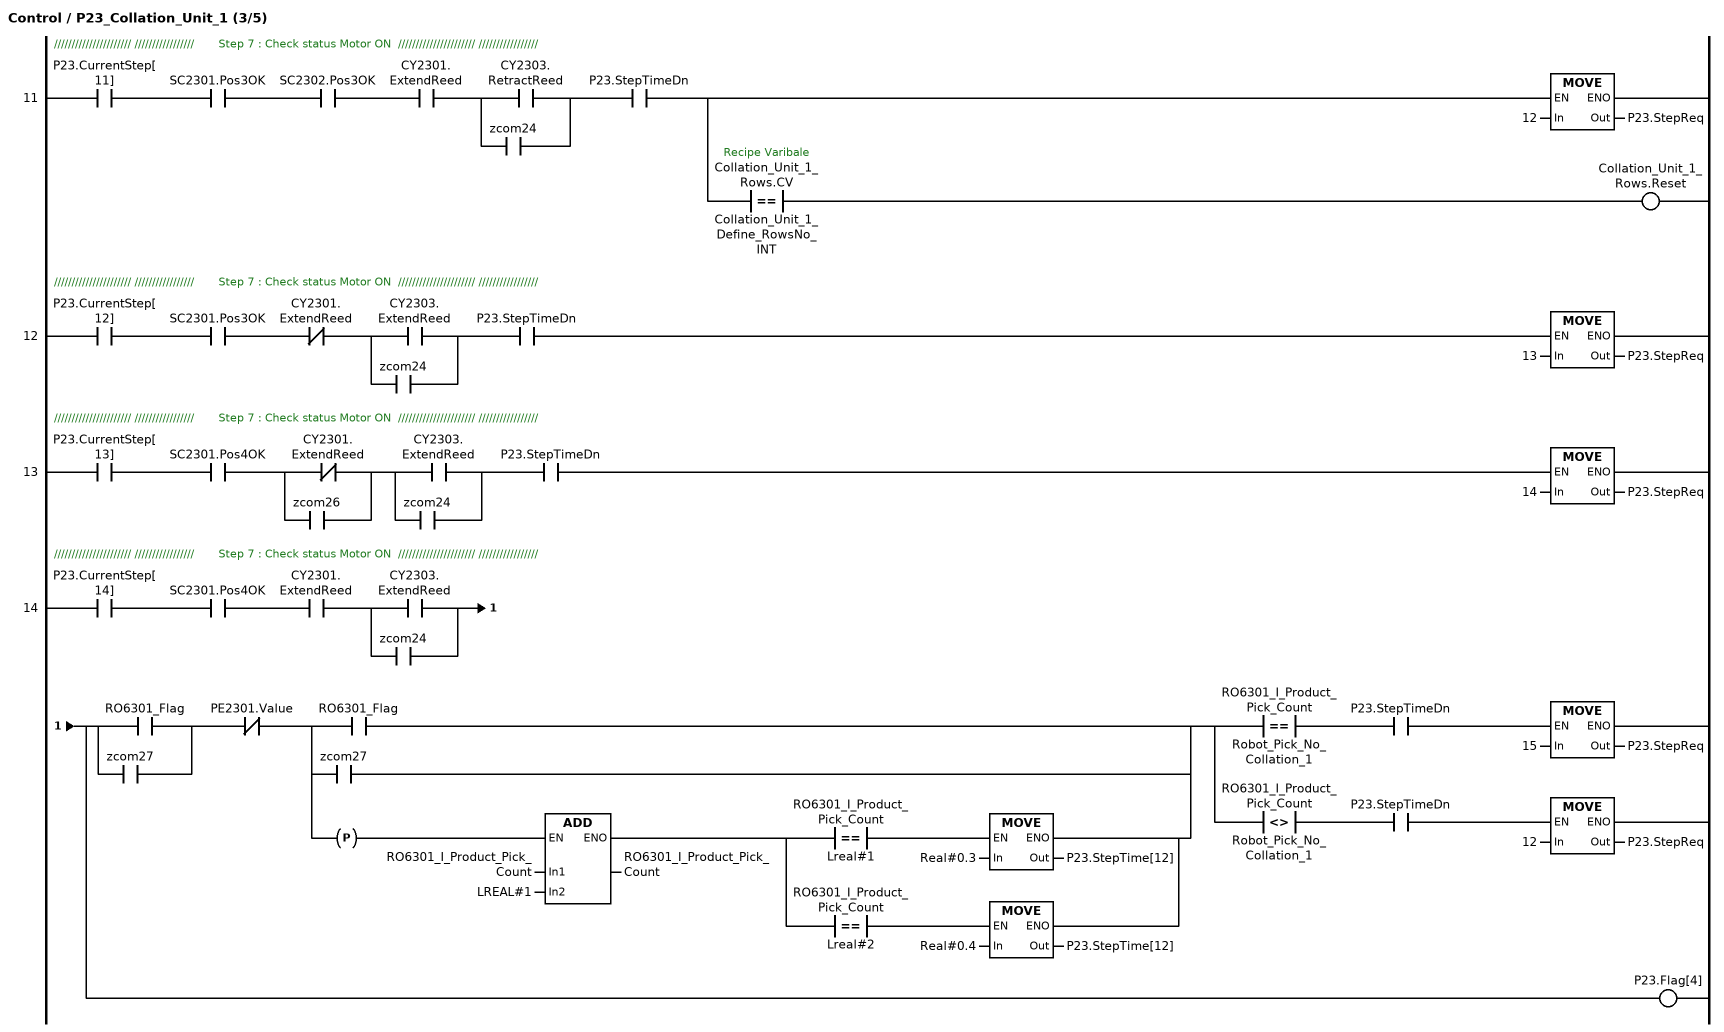
(* Rung 11: ////////////////////// /////////////////       Step 7 : Check status Motor ON  ////////////////////// ///////////////// *)
_p34 := P23.CurrentStep[11] AND SC2301.Pos3OK AND SC2302.Pos3OK AND CY2301.ExtendReed AND (CY2303.RetractReed OR zcom24) AND P23.StepTimeDn;
IF _p34 THEN P23.StepReq := 12; END_IF;
Collation_Unit_1_Rows.Reset := _p34 AND (Collation_Unit_1_Rows.CV = Collation_Unit_1_Define_RowsNo_INT);
(* Rung 12: ////////////////////// /////////////////       Step 7 : Check status Motor ON  ////////////////////// ///////////////// *)
IF P23.CurrentStep[12] AND SC2301.Pos3OK AND NOT CY2301.ExtendReed AND (CY2303.ExtendReed OR zcom24) AND P23.StepTimeDn THEN
    P23.StepReq := 13;
END_IF;
(* Rung 13: ////////////////////// /////////////////       Step 7 : Check status Motor ON  ////////////////////// ///////////////// *)
IF P23.CurrentStep[13] AND SC2301.Pos4OK AND (NOT CY2301.ExtendReed OR zcom26) AND (CY2303.ExtendReed OR zcom24) AND P23.StepTimeDn THEN
    P23.StepReq := 14;
END_IF;
(* Rung 14: ////////////////////// /////////////////       Step 7 : Check status Motor ON  ////////////////////// ///////////////// *)
_p35 := P23.CurrentStep[14] AND SC2301.Pos4OK AND CY2301.ExtendReed AND (CY2303.ExtendReed OR zcom24);
_p36 := _p35 AND (RO6301_Flag OR zcom27) AND NOT PE2301.Value;
_e37(CLK := _p36);
IF _e37.Q THEN RO6301_I_Product_Pick_Count := RO6301_I_Product_Pick_Count + LREAL#1; END_IF;
IF _e37.Q AND (RO6301_I_Product_Pick_Count = Lreal#1) THEN P23.StepTime[12] := Real#0.3; END_IF;
IF _e37.Q AND (RO6301_I_Product_Pick_Count = Lreal#2) THEN P23.StepTime[12] := Real#0.4; END_IF;
_p38 := (_p36 AND (RO6301_Flag OR zcom27)) OR (_e37.Q AND ((RO6301_I_Product_Pick_Count = Lreal#1) OR (RO6301_I_Product_Pick_Count = Lreal#2)));
IF _p38 AND (RO6301_I_Product_Pick_Count = Robot_Pick_No_Collation_1) AND P23.StepTimeDn THEN
    P23.StepReq := 15;
END_IF;
IF _p38 AND (RO6301_I_Product_Pick_Count <> Robot_Pick_No_Collation_1) AND P23.StepTimeDn THEN
    P23.StepReq := 12;
END_IF;
P23.Flag[4] := _p35;

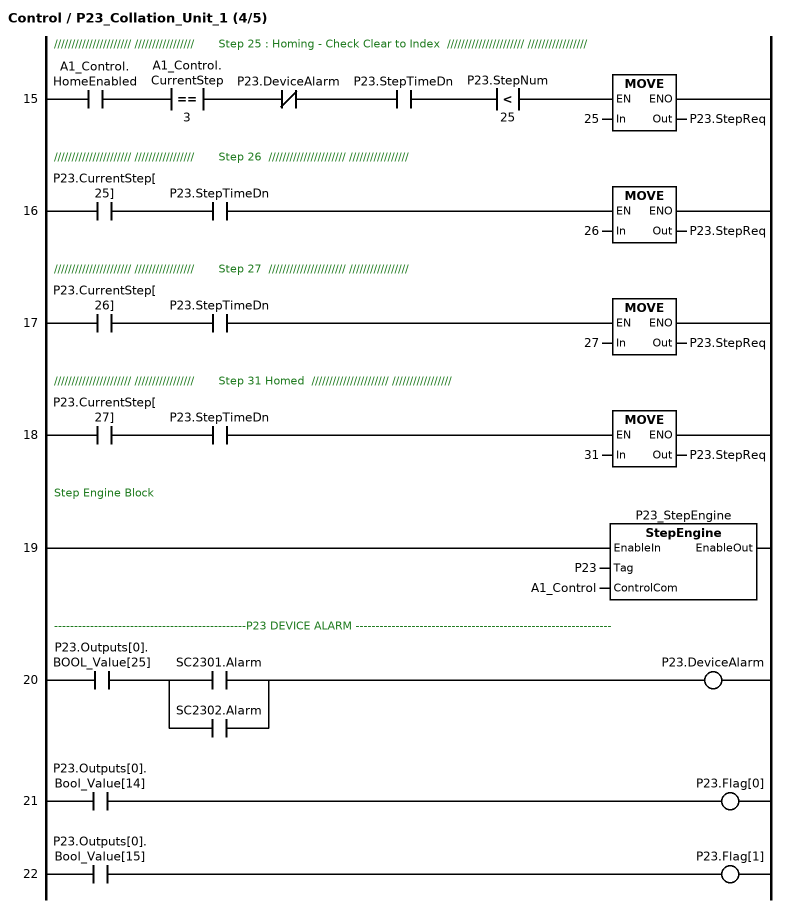
(* Rung 15: ////////////////////// /////////////////       Step 25 : Homing - Check Clear to Index  ////////////////////// ///////////////// *)
IF A1_Control.HomeEnabled AND (A1_Control.CurrentStep = 3) AND NOT P23.DeviceAlarm AND P23.StepTimeDn AND (P23.StepNum < 25) THEN
    P23.StepReq := 25;
END_IF;
(* Rung 16: ////////////////////// /////////////////       Step 26  ////////////////////// ///////////////// *)
IF P23.CurrentStep[25] AND P23.StepTimeDn THEN P23.StepReq := 26; END_IF;
(* Rung 17: ////////////////////// /////////////////       Step 27  ////////////////////// ///////////////// *)
IF P23.CurrentStep[26] AND P23.StepTimeDn THEN P23.StepReq := 27; END_IF;
(* Rung 18: ////////////////////// /////////////////       Step 31 Homed  ////////////////////// ///////////////// *)
IF P23.CurrentStep[27] AND P23.StepTimeDn THEN P23.StepReq := 31; END_IF;
(* Rung 19: Step Engine Block *)
P23_StepEngine(EnableIn := TRUE, Tag := P23, ControlCom := A1_Control);
(* Rung 20: ------------------------------------------------P23 DEVICE ALARM ---------------------------------------------------------------- *)
P23.DeviceAlarm := P23.Outputs[0].BOOL_Value[25] AND (SC2301.Alarm OR SC2302.Alarm);
(* Rung 21 *)
P23.Flag[0] := P23.Outputs[0].Bool_Value[14];
(* Rung 22 *)
P23.Flag[1] := P23.Outputs[0].Bool_Value[15];

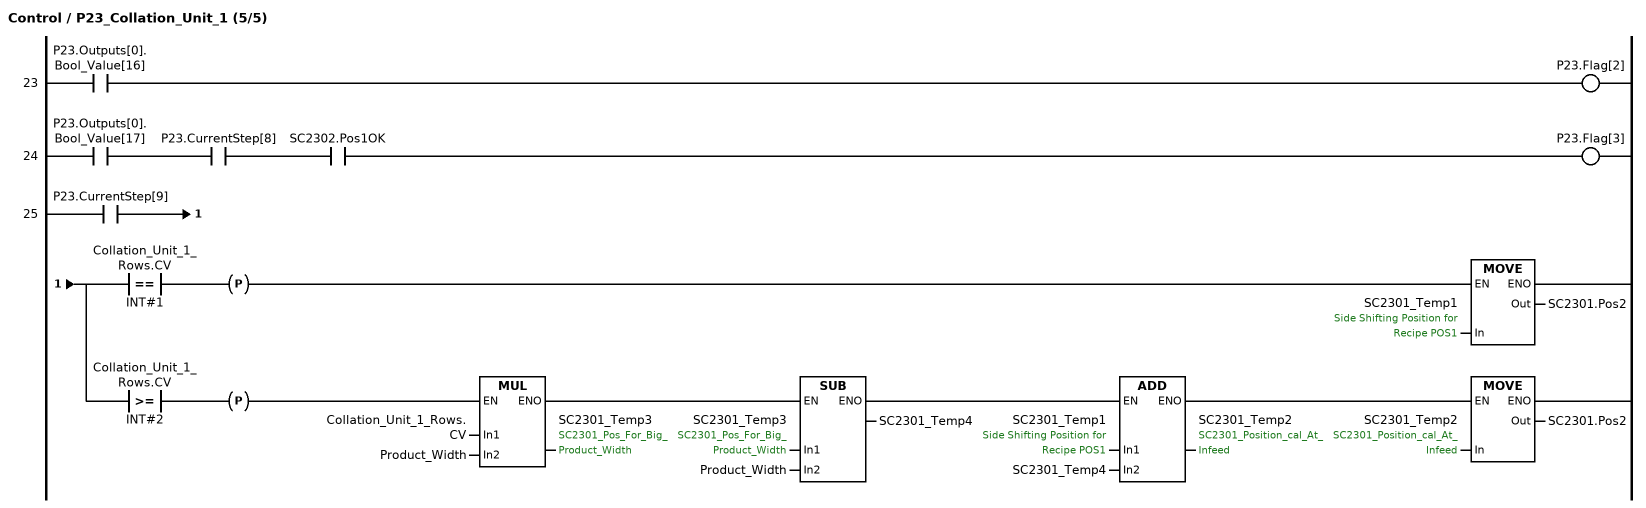
(* Rung 23 *)
P23.Flag[2] := P23.Outputs[0].Bool_Value[16];
(* Rung 24 *)
P23.Flag[3] := P23.Outputs[0].Bool_Value[17] AND P23.CurrentStep[8] AND SC2302.Pos1OK;
(* Rung 25 *)
_e39(CLK := P23.CurrentStep[9] AND (Collation_Unit_1_Rows.CV = INT#1));
IF _e39.Q THEN SC2301.Pos2 := SC2301_Temp1; END_IF;
_e40(CLK := P23.CurrentStep[9] AND (Collation_Unit_1_Rows.CV >= INT#2));
IF _e40.Q THEN
    SC2301_Temp3 := Collation_Unit_1_Rows.CV * Product_Width;
    SC2301_Temp4 := SC2301_Temp3 - Product_Width;
    SC2301_Temp2 := SC2301_Temp1 + SC2301_Temp4;
    SC2301.Pos2 := SC2301_Temp2;
END_IF;

(* Section P23a_Collation_Unit_2: ladder, written here as Structured Text *)

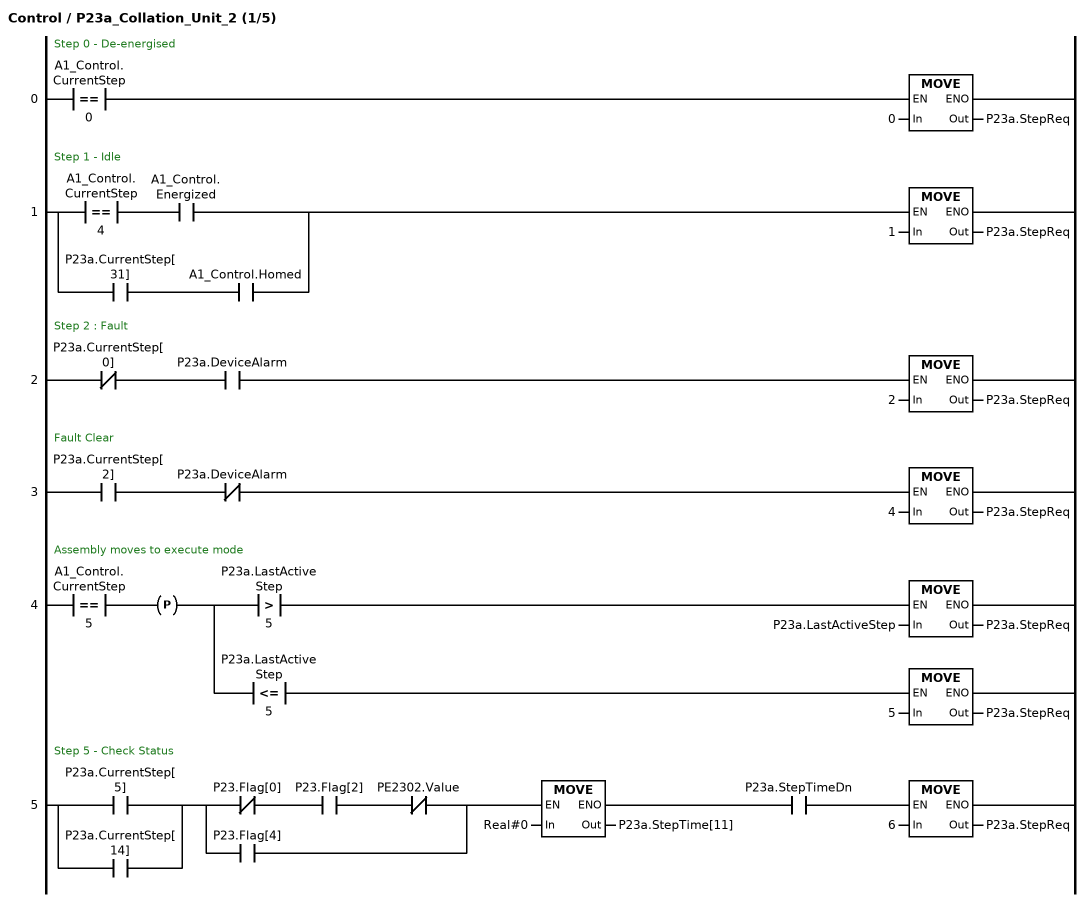
(* Rung 0: Step 0 - De-energised *)
IF A1_Control.CurrentStep = 0 THEN P23a.StepReq := 0; END_IF;
(* Rung 1: Step 1 - Idle *)
IF ((A1_Control.CurrentStep = 4) AND A1_Control.Energized) OR (P23a.CurrentStep[31] AND A1_Control.Homed) THEN
    P23a.StepReq := 1;
END_IF;
(* Rung 2: Step 2 : Fault *)
IF NOT P23a.CurrentStep[0] AND P23a.DeviceAlarm THEN P23a.StepReq := 2; END_IF;
(* Rung 3: Fault Clear *)
IF P23a.CurrentStep[2] AND NOT P23a.DeviceAlarm THEN P23a.StepReq := 4; END_IF;
(* Rung 4: Assembly moves to execute mode *)
_e41(CLK := A1_Control.CurrentStep = 5);
IF _e41.Q AND (P23a.LastActiveStep > 5) THEN P23a.StepReq := P23a.LastActiveStep; END_IF;
IF _e41.Q AND (P23a.LastActiveStep <= 5) THEN P23a.StepReq := 5; END_IF;
(* Rung 5: Step 5 - Check Status *)
_p42 := (P23a.CurrentStep[5] OR P23a.CurrentStep[14]) AND ((NOT P23.Flag[0] AND P23.Flag[2] AND NOT PE2302.Value) OR P23.Flag[4]);
IF _p42 THEN P23a.StepTime[11] := Real#0; END_IF;
IF _p42 AND P23a.StepTimeDn THEN P23a.StepReq := 6; END_IF;

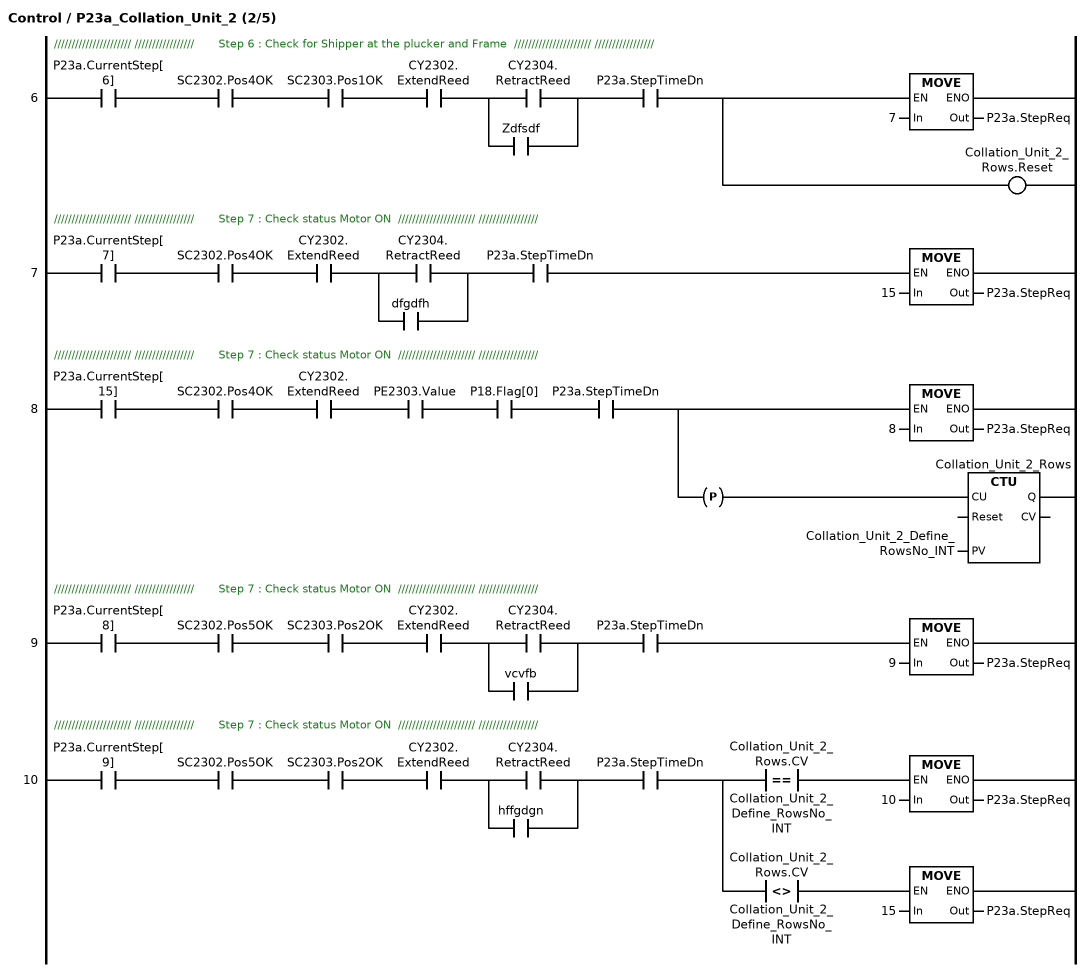
(* Rung 6: ////////////////////// /////////////////       Step 6 : Check for Shipper at the plucker and Frame  ////////////////////// ///////////////// *)
_p43 := P23a.CurrentStep[6] AND SC2302.Pos4OK AND SC2303.Pos1OK AND CY2302.ExtendReed AND (CY2304.RetractReed OR Zdfsdf) AND P23a.StepTimeDn;
IF _p43 THEN P23a.StepReq := 7; END_IF;
Collation_Unit_2_Rows.Reset := _p43;
(* Rung 7: ////////////////////// /////////////////       Step 7 : Check status Motor ON  ////////////////////// ///////////////// *)
IF P23a.CurrentStep[7] AND SC2302.Pos4OK AND CY2302.ExtendReed AND (CY2304.RetractReed OR dfgdfh) AND P23a.StepTimeDn THEN
    P23a.StepReq := 15;
END_IF;
(* Rung 8: ////////////////////// /////////////////       Step 7 : Check status Motor ON  ////////////////////// ///////////////// *)
_p44 := P23a.CurrentStep[15] AND SC2302.Pos4OK AND CY2302.ExtendReed AND PE2303.Value AND P18.Flag[0] AND P23a.StepTimeDn;
IF _p44 THEN P23a.StepReq := 8; END_IF;
_e45(CLK := _p44);
_e46(CLK := _e45.Q);
Collation_Unit_2_Rows(CU := _e46.Q, PV := Collation_Unit_2_Define_RowsNo_INT);
(* Rung 9: ////////////////////// /////////////////       Step 7 : Check status Motor ON  ////////////////////// ///////////////// *)
IF P23a.CurrentStep[8] AND SC2302.Pos5OK AND SC2303.Pos2OK AND CY2302.ExtendReed AND (CY2304.RetractReed OR vcvfb) AND P23a.StepTimeDn THEN
    P23a.StepReq := 9;
END_IF;
(* Rung 10: ////////////////////// /////////////////       Step 7 : Check status Motor ON  ////////////////////// ///////////////// *)
_p47 := P23a.CurrentStep[9] AND SC2302.Pos5OK AND SC2303.Pos2OK AND CY2302.ExtendReed AND (CY2304.RetractReed OR hffgdgn) AND P23a.StepTimeDn;
IF _p47 AND (Collation_Unit_2_Rows.CV = Collation_Unit_2_Define_RowsNo_INT) THEN
    P23a.StepReq := 10;
END_IF;
IF _p47 AND (Collation_Unit_2_Rows.CV <> Collation_Unit_2_Define_RowsNo_INT) THEN
    P23a.StepReq := 15;
END_IF;

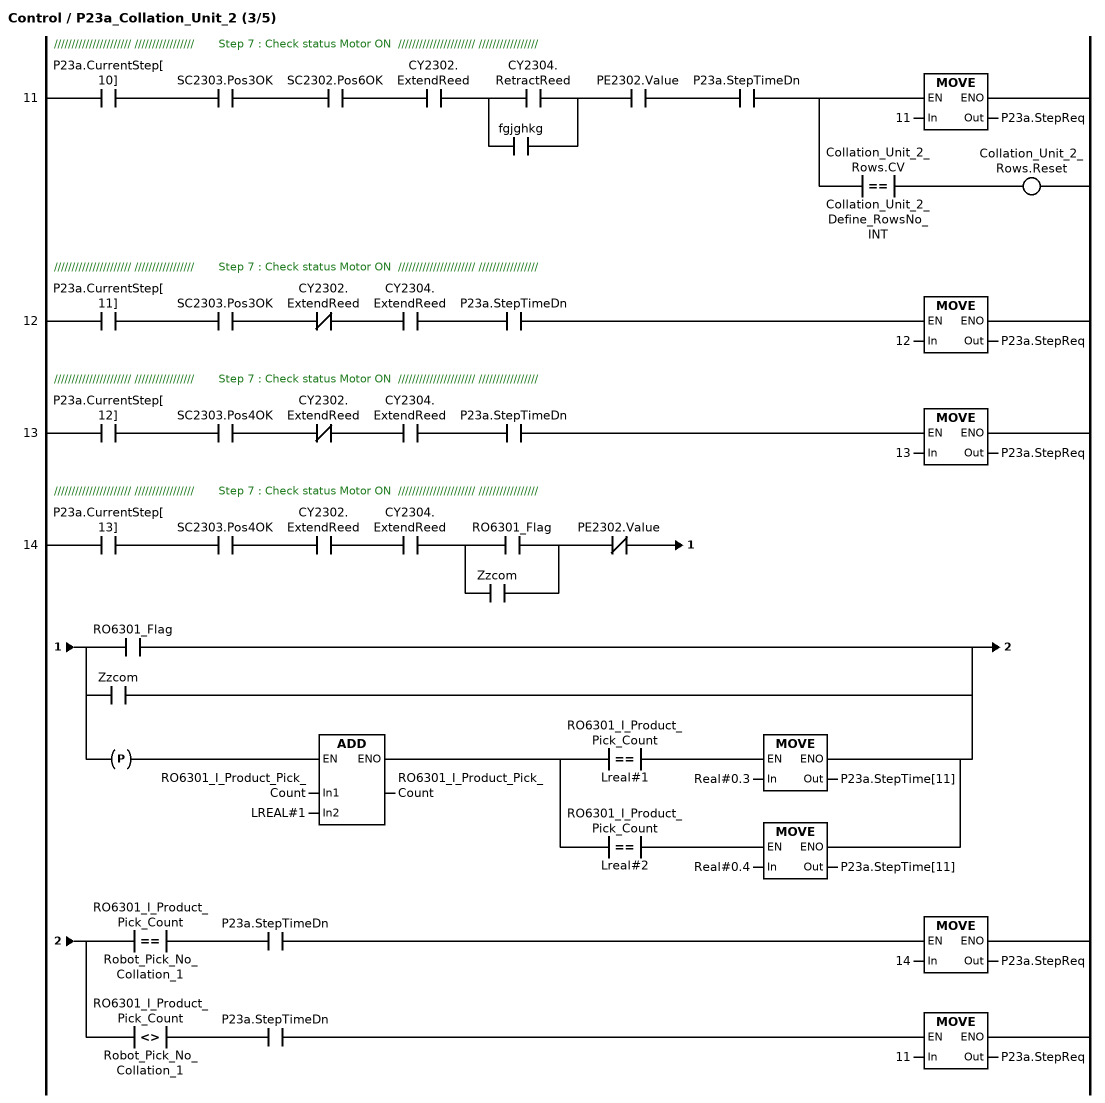
(* Rung 11: ////////////////////// /////////////////       Step 7 : Check status Motor ON  ////////////////////// ///////////////// *)
_p48 := P23a.CurrentStep[10] AND SC2303.Pos3OK AND SC2302.Pos6OK AND CY2302.ExtendReed AND (CY2304.RetractReed OR fgjghkg) AND PE2302.Value AND P23a.StepTimeDn;
IF _p48 THEN P23a.StepReq := 11; END_IF;
Collation_Unit_2_Rows.Reset := _p48 AND (Collation_Unit_2_Rows.CV = Collation_Unit_2_Define_RowsNo_INT);
(* Rung 12: ////////////////////// /////////////////       Step 7 : Check status Motor ON  ////////////////////// ///////////////// *)
IF P23a.CurrentStep[11] AND SC2303.Pos3OK AND NOT CY2302.ExtendReed AND CY2304.ExtendReed AND P23a.StepTimeDn THEN
    P23a.StepReq := 12;
END_IF;
(* Rung 13: ////////////////////// /////////////////       Step 7 : Check status Motor ON  ////////////////////// ///////////////// *)
IF P23a.CurrentStep[12] AND SC2303.Pos4OK AND NOT CY2302.ExtendReed AND CY2304.ExtendReed AND P23a.StepTimeDn THEN
    P23a.StepReq := 13;
END_IF;
(* Rung 14: ////////////////////// /////////////////       Step 7 : Check status Motor ON  ////////////////////// ///////////////// *)
_p49 := P23a.CurrentStep[13] AND SC2303.Pos4OK AND CY2302.ExtendReed AND CY2304.ExtendReed AND (RO6301_Flag OR Zzcom) AND NOT PE2302.Value;
_e50(CLK := _p49);
IF _e50.Q THEN RO6301_I_Product_Pick_Count := RO6301_I_Product_Pick_Count + LREAL#1; END_IF;
IF _e50.Q AND (RO6301_I_Product_Pick_Count = Lreal#1) THEN P23a.StepTime[11] := Real#0.3; END_IF;
IF _e50.Q AND (RO6301_I_Product_Pick_Count = Lreal#2) THEN P23a.StepTime[11] := Real#0.4; END_IF;
_p51 := (_p49 AND (RO6301_Flag OR Zzcom)) OR (_e50.Q AND ((RO6301_I_Product_Pick_Count = Lreal#1) OR (RO6301_I_Product_Pick_Count = Lreal#2)));
IF _p51 AND (RO6301_I_Product_Pick_Count = Robot_Pick_No_Collation_1) AND P23a.StepTimeDn THEN
    P23a.StepReq := 14;
END_IF;
IF _p51 AND (RO6301_I_Product_Pick_Count <> Robot_Pick_No_Collation_1) AND P23a.StepTimeDn THEN
    P23a.StepReq := 11;
END_IF;

